// TIA Portal V17 export
// export: Created 2025-03-13T10:31:44.9251261Z, ExportSetting WithDefaults, DisplayName Totally Integrated Automation Portal, DisplayVersion V17 Update 8, DisplayName TIA Portal Openness, DisplayVersion V17 Update 8, DisplayName TIA Portal Version Control Interface, DisplayVersion V17, DisplayName SINAMICS Startdrive Advanced, DisplayVersion V17 SP2, DisplayName SINAMICS Startdrive G110M, G120, G120C, G120D, G120P, G115D, DisplayVersion V17 SP2, DisplayName SINAMICS Startdrive G130, G150, S120, S150, SINAMICS MV, S210, DisplayVersion V17 SP2, DisplayName STEP 7 Professional, DisplayVersion V17 Update 8, DisplayName SINUMERIK ONE STEP 7 Toolbox, DisplayVersion V17 Update 12, DisplayName SINUMERIK 840D sl STEP 7 Toolbox, DisplayVersion V17 Update 12, DisplayName STEP 7 Safety, DisplayVersion V17 Update 6, DisplayName WinCC Advanced, DisplayVersion V17 Update 8
TYPE "MPP_INPUTS"
// stored: IsFailsafeCompliant false
   STRUCT
      I_S59_E_STOP_OVERRIDE : Bool;   // S59 - S11 HAND HELD PANEL ENABLE / S59 - S11 EMERGENCY STOP OVERRIDE
      I_S60 : Bool;   // S60 - S11 BA MODE ENABLE / S60 - EXTENSION KEY
      I_S62_HG_CONNECTION : Bool;   // S62 - XS12:13 HG CONNECTION
      I_F21 : Bool;   // F21 FUNCTION KEY - RESET
      I_WS1_1 : Bool;   // F1 FUNCTION KEY - CONTINUOUS CYCLE // BA WS1/1 / WS1/1 - CONTINUOUS CYCLE
      I_WS1_2 : Bool;   // F6 FUNCTION KEY - ONE CYCLE // BA WS1/2 / WS1/2 - SINGLE CYCLE
      I_WS1_3 : Bool;   // F11 FUNCTION KEY - STEP BY STEP CYCLE // BA WS1/3 / WS1/3 - STEP BY STEP CYCLE
      I_WS1_4 : Bool;   // F16 FUNCTION KEY - SETUP // BA WS1/4 / WS1/4 - SETUP
      I_S1 : Bool;   // MPP483 KEY - CONTROL ON / S1 KEY - CONTROL ON
      I_S2 : Bool;   // MPP483 KEY - START / S2 KEY - START
      I_S3 : Bool;   // MPP483 KEY - HOME POSITION / S3 KEY - HOME POSITION
      I_S4 : Bool;   // MPP483 KEY - RESET FAULT / S4 KEY - RESET FAULT
      I_S51 : Bool;   // S51 EXTENSION KEY - / S51 - EXTENSION KEY
      I_S14 : Bool;   // S5 CUSTOMER KEY - / S14 - USER KEY
      I_WS4_KEY_POS_0 : Bool;   // MPP483 KEY - POSITION 0 / WS4 KEY - POSITION 0
      I_S15 : Bool;   // MPP483 KEY - / S15 KEY - USER KEY
      I_WS5_1_RAP_TRAV_OVERR : Bool;   // WS5/1 - RAPID TRAVERSE OVERRIDE
      I_WS5_2_RAP_TRAV_OVERR : Bool;   // WS5/2 - RAPID TRAVERSE OVERRIDE
      I_WS5_4_RAP_TRAV_OVERR : Bool;   // WS5/4 - RAPID TRAVERSE OVERRIDE
      I_WS5_8_RAP_TRAV_OVERR : Bool;   // WS5/8 - RAPID TRAVERSE OVERRIDE
      I_S61 : Bool;   // S61 - SR KEY / S61 - EXTENSION KEY
      I_WS4_KEY_POS_1 : Bool;   // WS4 KEY - POSITION 1
      I_WS4_KEY_POS_2 : Bool;   // WS4 KEY - POSITION 2
      I_WS4_KEY_POS_3 : Bool;   // WS4 KEY - POSITION 3
      I_S52 : Bool;   // S52 EXTENSION KEY - / S52 - EXTENSION KEY
      I_S7 : Bool;   // MPP483 KEY - CONTROL OFF / S7 KEY - CONTROL OFF
      I_S8 : Bool;   // MPP483 KEY - REQUEST STOP END OF CYCLE / S8 KEY - REQUEST STOP END OF CYCLE
      I_S9 : Bool;   // MPP483 KEY - IMMEDIATE STOP / S9 KEY - IMMEDIATE STOP
      I_S10 : Bool;   // MPP483 KEY - UNLOCK SAFETY DOORS / S10 KEY - UNLOCK SAFETY DOORS
      I_S13 : Bool;   // S11 - EMERGENCY STOP / S13 - EMERGENCY STOP
      I_S53 : Bool;   // S53 EXTENSION KEY - / S53 - EXTENSION KEY
      I_3_7 : Bool;   // NOT USED
      I_DT1 : Bool;   // DT1 - DIRECT CONTROL KEY / DT1 - DIRECT KEY
      I_DT2 : Bool;   // DT2 - DIRECT CONTROL KEY / DT2 - DIRECT KEY
      I_DT3 : Bool;   // DT3 - DIRECT CONTROL KEY / DT3 - DIRECT KEY
      I_DT4 : Bool;   // DT4 - DIRECT CONTROL KEY / DT4 - DIRECT KEY
      I_DT5 : Bool;   // DT5 - DIRECT CONTROL KEY / DT5 - DIRECT KEY
      I_DT6 : Bool;   // DT6 - DIRECT CONTROL KEY / DT6 - DIRECT KEY
      I_DT7 : Bool;   // DT7 - DIRECT CONTROL KEY / DT7 - DIRECT KEY
      I_DT8 : Bool;   // DT8 - DIRECT CONTROL KEY / DT8 - DIRECT KEY
      I_DT9 : Bool;   // DT9 - DIRECT CONTROL KEY / DT9 - DIRECT KEY
      I_DT10 : Bool;   // DT10 - DIRECT CONTROL KEY / DT10 - DIRECT KEY
      I_DT11 : Bool;   // DT11 - DIRECT CONTROL KEY / DT11 - DIRECT KEY
      I_DT12 : Bool;   // DT12 - DIRECT CONTROL KEY / DT12 - DIRECT KEY
      I_DT13 : Bool;   // DT13 - DIRECT CONTROL KEY / DT13 - DIRECT KEY
      I_DT14 : Bool;   // DT14 - DIRECT CONTROL KEY / DT14 - DIRECT KEY
      I_DT15 : Bool;   // DT15 - DIRECT CONTROL KEY / DT15 - DIRECT KEY
      I_DT16 : Bool;   // DT16 - DIRECT CONTROL KEY / DT16 - DIRECT KEY
      I_WS3_1_SPIND_OVERR : Bool;   // WS3/1 - SPINDLE OVERRIDE
      I_WS3_2_SPIND_OVERR : Bool;   // WS3/2 - SPINDLE OVERRIDE
      I_WS3_4_SPIND_OVERR : Bool;   // WS3/4 - SPINDLE OVERRIDE
      I_WS3_8_SPIND_OVERR : Bool;   // WS3/8 - SPINDLE OVERRIDE
      I_S57 : Bool;   // S57 EXTENSION KEY - / S57 - EXTENSION KEY
      I_S58 : Bool;   // S58 EXTENSION KEY - / S58 - EXTENSION KEY
      I_6_6 : Bool;   // NOT USED
      I_6_7 : Bool;   // NOT USED
      I_WS2_1_FEED_OVERR : Bool;   // WS2/1 - FEEDRATE OVERRIDE
      I_WS2_2_FEED_OVERR : Bool;   // WS2/2 - FEEDRATE OVERRIDE
      I_WS2_4_FEED_OVERR : Bool;   // WS2/4 - FEEDRATE OVERRIDE
      I_WS2_8_FEED_OVERR : Bool;   // WS2/8 - FEEDRATE OVERRIDE
      I_WS2_16_FEED_OVERR : Bool;   // WS2/16 - FEEDRATE OVERRIDE
      I_S54 : Bool;   // S54 EXTENSION KEY - / S54 - EXTENSION KEY
      I_S55 : Bool;   // S55 EXTENSION KEY - / S55 - EXTENSION KEY
      I_S56 : Bool;   // S56 EXTENSION KEY - / S56 - EXTENSION KEY
      I_F1 : Bool;   // F1 FUNCTION KEY - CONTINUOUS CYCLE
      I_F2 : Bool;   // F2 FUNCTION KEY - AUTOMATIC MODE
      I_F3 : Bool;   // F3 FUNCTION KEY - SINGLE BLOCK
      I_F4 : Bool;   // F4 FUNCTION KEY - NC STOP
      I_F5 : Bool;   // F5 FUNCTION KEY - NC START
      I_F6 : Bool;   // F6 FUNCTION KEY - ONE CYCLE / F6 FUNCTION KEY - SINGLE CYCLE
      I_F7 : Bool;   // F7 FUNCTION KEY - MDA MODE
      I_F8 : Bool;   // F8 FUNCTION KEY - NEXT AXES
      I_F9 : Bool;   // F9 FUNCTION KEY - FEEDRATE STOP
      I_F10 : Bool;   // F10 FUNCTION KEY - FEEDRATE START
      I_F11 : Bool;   // F11 FUNCTION KEY - STEP BY STEP CYCLE
      I_F12 : Bool;   // F12 FUNCTION KEY - JOG MODE
      I_F13 : Bool;   // F13 FUNCTION KEY - (X1 - W) AXES / F13 FUNCTION KEY - (X11 - W) AXES
      I_F14 : Bool;   // F14 FUNCTION KEY - (Y1 - E) AXES / F14 FUNCTION KEY - (Y11 - E) AXES
      I_F15 : Bool;   // F15 FUNCTION KEY - Z11 AXIS
      I_F16 : Bool;   // F16 FUNCTION KEY - SETUP MODE
      I_F17 : Bool;   // F17 FUNCTION KEY - REFERENCE POINT MODE
      I_F18 : Bool;   // F18 FUNCTION KEY - (A - U1 - C) AXES / F18 FUNCTION KEY - (A11 - U11 - C) AXES
      I_F19 : Bool;   // F18 FUNCTION KEY - B AXIS / F19 FUNCTION KEY - B AXIS
      I_F20 : Bool;   // F18 FUNCTION KEY - (Q1 - Z12) AXES / F20 FUNCTION KEY - (Q11 - Z12) AXES
      I_F22 : Bool;   // F22 FUNCTION KEY - INCREMENTAL MODE
      I_F23 : Bool;   // F23 FUNCTION KEY - MINUS DIRECTION
      I_F24 : Bool;   // F24 FUNCTION KEY - RAPID
      I_F25 : Bool;   // F25 FUNCTION KEY - PLUS DIRECTION
      I_BYTE_11 : Byte;   // RESERVED / RESERVE
      I_WS2_1_FEED_OVERRIDE : Bool;   // WS2/1 - FEEDRATE OVERRIDE
      I_WS2_2_FEED_OVERRIDE : Bool;   // WS2/2 - FEEDRATE OVERRIDE
      I_WS2_4_FEED_OVERRIDE : Bool;   // WS2/4 - FEEDRATE OVERRIDE
      I_WS2_8_FEED_OVERRIDE : Bool;   // WS2/8 - FEEDRATE OVERRIDE
      I_WS2_16_FEED_OVERRIDE : Bool;   // WS2/16 - FEEDRATE OVERRIDE
      I_12_5 : Bool;   // NOT USED
      I_12_6 : Bool;   // NOT USED
      I_12_7 : Bool;   // NOT USED
      I_WS3_1_SPIND_OVERRIDE : Bool;   // WS3/1 - SPINDLE OVERRIDE
      I_WS3_2_SPIND_OVERRIDE : Bool;   // WS3/2 - SPINDLE OVERRIDE
      I_WS3_4_SPIND_OVERRIDE : Bool;   // WS3/4 - SPINDLE OVERRIDE
      I_WS3_8_SPIND_OVERRIDE : Bool;   // WS3/8 - SPINDLE OVERRIDE
      I_WS3_16_SPIND_OVERRIDE : Bool;   // WS3/16 - SPINDLE OVERRIDE
      I_13_5 : Bool;   // NOT USED
      I_13_6 : Bool;   // NOT USED
      I_13_7 : Bool;   // NOT USED
      HANDWHEEL_1_COUNTER_READ : Int;   // HANDWHEEL 1 - COUNTER STATUS / HANDWHEEL 1 - COUNTER READING
      HANDWHEEL_2_COUNTER_READ : Int;   // HANDWHEEL 2 - COUNTER STATUS / HANDWHEEL 2 - COUNTER READING
   END_STRUCT;
END_TYPE
